(* IEC 61131-3 sources: AXOpen/src/components.ur.robotics/ctrl/src/AxoUrCb3/v_3_x_x, 1 file *)

(* ---- AxoUrCb3.st ---- *)
USING AXOpen.Core;
USING AXOpen.Messaging;
USING AXOpen.Messaging.Static;
USING AXOpen.Components.Robotics;
USING AXOpen.Components.Abstractions.Robotics;
USING Siemens.Simatic.Hardware.Utilities;

NAMESPACE AXOpen.Components.Ur.Robotics.v_3_x_x
    {S7.extern=ReadWrite}
    CLASS AxoUrCb3 EXTENDS AXOpen.Core.AxoComponent IMPLEMENTS AXOpen.Components.Abstractions.Robotics.IAxoRobotics
        VAR PRIVATE
            _infoTimer              :   AXOpen.Timers.OnDelayTimer;
            _errorTimer             :   AXOpen.Timers.OnDelayTimer;
            _context                :   IAxoContext;
            _stopTasksAreActive     :   BOOL;
            _stopType               :   eAxoRoboticsStopType;
            _someTaskIsActive       :   BOOL;

            _initHwCheckDone        :   BOOL;
            _retval                 :   WORD;
            _geoAddr                :   GeoAddr;
            _outHwid                :   UINT;
            _blink                  :   AXOpen.Timers.AxoBlinker;
            _inputsAddress          :   UDINT;
            _inputsCount            :   UINT;
            _outputsAddress         :   UDINT;
            _outputsCount           :   UINT;
        END_VAR

        VAR PUBLIC //HEADER

        END_VAR

        VAR PUBLIC //Tasks
            {#ix-attr:[Container(Layout.Wrap)]}
            {#ix-attr:[ComponentDetails("Tasks")]}
            {#ix-set:AttributeName = "<#Restore#>"}
            RestoreTask : AxoTask;

            {#ix-attr:[ComponentDetails("Tasks")]}
            {#ix-set:AttributeName = "<#Power On Task#>"}
            PowerOnTask : AxoTask;

            {#ix-attr:[Container(Layout.Wrap)]}
            {#ix-attr:[ComponentDetails("Tasks")]}
            {#ix-set:AttributeName = "<#Start at main#>"}
            StartAtMainTask : AxoTask;

            {#ix-attr:[ComponentDetails("Tasks")]}
            {#ix-set:AttributeName = "<#Start motors and program#>"}
            StartMotorsAndProgramTask : AxoTask;

            {#ix-attr:[ComponentDetails("Tasks")]}
            {#ix-set:AttributeName = "<#Stop movements#>"}
            StopMovementsTask : AxoTask;

            {#ix-attr:[ComponentDetails("Tasks")]}
            {#ix-set:AttributeName = "<#Stop movements and program#>"}
            StopMovementsAndProgramTask : AxoTask;

            {#ix-attr:[ComponentDetails("Tasks")]}
            {#ix-set:AttributeName = "<#Start movements with extended parameters#>"}
            StartMovementsTask : AxoTask;

            {#ix-attr:[ComponentDetails("Tasks")]}
            {#ix-set:AttributeName = "<#Start movements with extended parameters#>"}
            MovementParameters : AXOpen.Components.Abstractions.Robotics.AxoRoboticsMovementsParams;
        END_VAR

        VAR PUBLIC //CONFIG
            {#ix-attr:[Container(Layout.Stack)]}
            {#ix-attr:[ComponentDetails("Config")]}
            {#ix-attr:[ReadOnly()]}
            Config  :   AxoUrRobotics_Config;
        END_VAR

        VAR PUBLIC //STATUS
            {#ix-attr:[Container(Layout.Stack)]}
            {#ix-attr:[ComponentDetails("Status")]}
            {#ix-attr:[ReadOnly()]}
            Status         :   AxoUrRobotics_Component_Status;
            {#ix-attr:[ComponentDetails("Status")]}
            {#ix-attr:[ReadOnly()]}
            {#ix-set:AttributeName = "<#Power progress#>"}
            _power_progress  :   INT := 0;
            {#ix-attr:[ComponentDetails("Status")]}
            {#ix-attr:[ReadOnly()]}
            {#ix-set:AttributeName = "<#Movement progress#>"}
            _movement_progress  :   INT := 0;
            Messenger           :   AXOpen.Messaging.Static.AxoMessenger;
            TaskMessenger       :   AXOpen.Messaging.Static.AxoMessenger;
        END_VAR

        VAR PUBLIC //Hardware signals
            {#ix-attr:[ComponentDetails("Hardware signals")]}
            {#ix-attr:[Container(Layout.Wrap)]}
            {#ix-attr:[Group(GroupLayout.GroupBox)]}
            {#ix-set:AttributeName = "<#Inputs#>"}
            {#ix-attr:[ReadOnly()]}
            Inputs              :   AxoUrRobotics_State;
            {#ix-attr:[ComponentDetails("Hardware signals")]}
            {#ix-attr:[Container(Layout.Wrap)]}
            {#ix-attr:[Group(GroupLayout.GroupBox)]}
            {#ix-set:AttributeName = "<#Outputs#>"}
            {#ix-attr:[ReadOnly()]}
            Outputs              :   AxoUrRobotics_Control;
        END_VAR

        VAR PUBLIC //HardwareDiagnostics
            {#ix-attr:[Container(Layout.Stack)]}
            {#ix-attr:[ComponentDetails("Hardware diagnostics")]}
            {#ix-set:AttributeName = "<#Update diagnostics#>"}
            HardwareDiagnosticsTask :   AXOpen.Io.AxoHardwareDiagnostics;
            {#ix-attr:[ComponentDetails("Hardware diagnostics")]}
            {#ix-set:AttributeName = "<#Reboot controller#>"}
            RebootControllerTask : AxoRemoteTask ;
        END_VAR

        ///<summary>
        /// Runs tasks and logic of this component.
        /// >[!IMPORTANT] This method must or one of its overloads be called cyclically.
        ///</summary>
        METHOD PUBLIC Run
            VAR_INPUT
                inParent        :   IAxoObject;
                hwID            :   UINT;
                refPowerOnPulse :   REF_TO BOOL;
            END_VAR
            VAR
                _word : WORD;
                _dword: DWORD;
                _retVal : WORD;
                _data : ARRAY[0..103] OF BYTE;
                _data24 : ARRAY[0..23] OF BYTE;
                _data100 : ARRAY[0..99] OF BYTE;
            END_VAR

            SUPER.Run(inParent);

            Messenger.Serve(THIS);

            IF NOT _initHwCheckDone THEN
                IF inParent = NULL THEN
                    Messenger.Activate(UINT#700, eAxoMessageCategory#ProgrammingError);
                    Status.Error.Id := UINT#700;
                    RETURN;
                END_IF;
                Config.HWIDs.HwId_Device  := hwID;
                IF Config.HWIDs.HwId_Device = UINT#0 THEN
                    Messenger.Activate(UINT#701, eAxoMessageCategory#ProgrammingError);
                    Status.Error.Id := UINT#701;
                    RETURN;
                END_IF;

                _retval := ReadSlotFromHardwareID(hardwareID := Config.HWIDs.HwId_Device, geoAddr :=_geoAddr);
                IF _retval = WORD#8090 THEN
                    Messenger.Activate(UINT#702,eAxoMessageCategory#Error);
                    Status.Error.Id := UINT#702;
                    RETURN;
                END_IF;

                //******************Slot 1*****************//
                _geoAddr.Slot   :=  UINT#1;
                _geoAddr.HardwareType := UINT#4; // (4-Module)
                _retval := ReadHardwareIDFromSlot(geoAddr := _geoAddr, hardwareID => _outHwid);
                IF Config.HWIDs.HwId_AxoUrRobotics_T2O_State = UINT#0 THEN
                    Messenger.Activate(UINT#710,eAxoMessageCategory#Error);
                    Status.Error.Id := UINT#710;
                    RETURN;
                END_IF;
                IF _retval = WORD#8091 THEN
                    Messenger.Activate(UINT#711,eAxoMessageCategory#Error);
                    Status.Error.Id := UINT#711;
                    RETURN;
                END_IF;
                IF _retval = WORD#8094 THEN
                    Messenger.Activate(UINT#712,eAxoMessageCategory#Error);
                    Status.Error.Id := UINT#712;
                    RETURN;
                END_IF;
                IF _retval = WORD#8095 THEN
                    Messenger.Activate(UINT#713,eAxoMessageCategory#Error);
                    Status.Error.Id := UINT#713;
                    RETURN;
                END_IF;
                IF _retval = WORD#8096 THEN
                    Messenger.Activate(UINT#714,eAxoMessageCategory#Error);
                    Status.Error.Id := UINT#714;
                    RETURN;
                END_IF;
                IF _retval = WORD#8097 THEN
                    Messenger.Activate(UINT#715,eAxoMessageCategory#Error);
                    Status.Error.Id := UINT#715;
                    RETURN;
                END_IF;
                ReadHardwareIOAddress(hardwareID := (Config.HWIDs.HwId_AxoUrRobotics_T2O_State) , inputStartAddress => _inputsAddress , inputCount => _inputsCount , outputStartAddress => _outputsAddress , outputCount => _outputsCount);
                IF _inputsCount <> UINT#32 OR _outputsCount <> UINT#0 THEN
                    Messenger.Activate(UINT#716,eAxoMessageCategory#Error);
                    Status.Error.Id := UINT#716;
                    RETURN;
                END_IF;
                //******************Slot 2*****************//
                _geoAddr.Slot   :=  UINT#2;
                _geoAddr.HardwareType := UINT#4; // (4-Module)
                _retval := ReadHardwareIDFromSlot(geoAddr := _geoAddr, hardwareID => _outHwid);
                IF Config.HWIDs.HwId_AxoUrRobotics_T2O_IO = UINT#0 THEN
                    Messenger.Activate(UINT#720,eAxoMessageCategory#Error);
                    Status.Error.Id := UINT#720;
                    RETURN;
                END_IF;
                IF _retval = WORD#8091 THEN
                    Messenger.Activate(UINT#721,eAxoMessageCategory#Error);
                    Status.Error.Id := UINT#721;
                    RETURN;
                END_IF;
                IF _retval = WORD#8094 THEN
                    Messenger.Activate(UINT#722,eAxoMessageCategory#Error);
                    Status.Error.Id := UINT#722;
                    RETURN;
                END_IF;
                IF _retval = WORD#8095 THEN
                    Messenger.Activate(UINT#723,eAxoMessageCategory#Error);
                    Status.Error.Id := UINT#723;
                    RETURN;
                END_IF;
                IF _retval = WORD#8096 THEN
                    Messenger.Activate(UINT#724,eAxoMessageCategory#Error);
                    Status.Error.Id := UINT#724;
                    RETURN;
                END_IF;
                IF _retval = WORD#8097 THEN
                    Messenger.Activate(UINT#725,eAxoMessageCategory#Error);
                    Status.Error.Id := UINT#725;
                    RETURN;
                END_IF;
                ReadHardwareIOAddress(hardwareID := (Config.HWIDs.HwId_AxoUrRobotics_T2O_IO) , inputStartAddress => _inputsAddress , inputCount => _inputsCount , outputStartAddress => _outputsAddress , outputCount => _outputsCount);
                IF _inputsCount <> UINT#68 OR _outputsCount <> UINT#0 THEN
                    Messenger.Activate(UINT#726,eAxoMessageCategory#Error);
                    Status.Error.Id := UINT#726;
                    RETURN;
                END_IF;
                //******************Slot 3*****************//
                _geoAddr.Slot   :=  UINT#3;
                _geoAddr.HardwareType := UINT#4; // (4-Module)
                _retval := ReadHardwareIDFromSlot(geoAddr := _geoAddr, hardwareID => _outHwid);
                IF Config.HWIDs.HwId_AxoUrRobotics_T2O_Joints = UINT#0 THEN
                    Messenger.Activate(UINT#730,eAxoMessageCategory#Error);
                    Status.Error.Id := UINT#730;
                    RETURN;
                END_IF;
                IF _retval = WORD#8091 THEN
                    Messenger.Activate(UINT#731,eAxoMessageCategory#Error);
                    Status.Error.Id := UINT#731;
                    RETURN;
                END_IF;
                IF _retval = WORD#8094 THEN
                    Messenger.Activate(UINT#732,eAxoMessageCategory#Error);
                    Status.Error.Id := UINT#732;
                    RETURN;
                END_IF;
                IF _retval = WORD#8095 THEN
                    Messenger.Activate(UINT#733,eAxoMessageCategory#Error);
                    Status.Error.Id := UINT#733;
                    RETURN;
                END_IF;
                IF _retval = WORD#8096 THEN
                    Messenger.Activate(UINT#734,eAxoMessageCategory#Error);
                    Status.Error.Id := UINT#734;
                    RETURN;
                END_IF;
                IF _retval = WORD#8097 THEN
                    Messenger.Activate(UINT#735,eAxoMessageCategory#Error);
                    Status.Error.Id := UINT#735;
                    RETURN;
                END_IF;
                ReadHardwareIOAddress(hardwareID := (Config.HWIDs.HwId_AxoUrRobotics_T2O_Joints) , inputStartAddress => _inputsAddress , inputCount => _inputsCount , outputStartAddress => _outputsAddress , outputCount => _outputsCount);
                IF _inputsCount <> UINT#104 OR _outputsCount <> UINT#0 THEN
                    Messenger.Activate(UINT#736,eAxoMessageCategory#Error);
                    Status.Error.Id := UINT#736;
                    RETURN;
                END_IF;
                //******************Slot 4*****************//
                _geoAddr.Slot   :=  UINT#4;
                _geoAddr.HardwareType := UINT#4; // (4-Module)
                _retval := ReadHardwareIDFromSlot(geoAddr := _geoAddr, hardwareID => _outHwid);
                IF Config.HWIDs.HwId_AxoUrRobotics_T2O_TCP = UINT#0 THEN
                    Messenger.Activate(UINT#740,eAxoMessageCategory#Error);
                    Status.Error.Id := UINT#740;
                    RETURN;
                END_IF;
                IF _retval = WORD#8091 THEN
                    Messenger.Activate(UINT#741,eAxoMessageCategory#Error);
                    Status.Error.Id := UINT#741;
                    RETURN;
                END_IF;
                IF _retval = WORD#8094 THEN
                    Messenger.Activate(UINT#742,eAxoMessageCategory#Error);
                    Status.Error.Id := UINT#742;
                    RETURN;
                END_IF;
                IF _retval = WORD#8095 THEN
                    Messenger.Activate(UINT#743,eAxoMessageCategory#Error);
                    Status.Error.Id := UINT#743;
                    RETURN;
                END_IF;
                IF _retval = WORD#8096 THEN
                    Messenger.Activate(UINT#744,eAxoMessageCategory#Error);
                    Status.Error.Id := UINT#744;
                    RETURN;
                END_IF;
                IF _retval = WORD#8097 THEN
                    Messenger.Activate(UINT#745,eAxoMessageCategory#Error);
                    Status.Error.Id := UINT#745;
                    RETURN;
                END_IF;
                ReadHardwareIOAddress(hardwareID := (Config.HWIDs.HwId_AxoUrRobotics_T2O_TCP) , inputStartAddress => _inputsAddress , inputCount => _inputsCount , outputStartAddress => _outputsAddress , outputCount => _outputsCount);
                IF _inputsCount <> UINT#76 OR _outputsCount <> UINT#0 THEN
                    Messenger.Activate(UINT#746,eAxoMessageCategory#Error);
                    Status.Error.Id := UINT#746;
                    RETURN;
                END_IF;
                //******************Slot 5*****************//
                _geoAddr.Slot   :=  UINT#5;
                _geoAddr.HardwareType := UINT#4; // (4-Module)
                _retval := ReadHardwareIDFromSlot(geoAddr := _geoAddr, hardwareID => _outHwid);
                IF Config.HWIDs.HwId_AxoUrRobotics_T2O_General_Purpose_Bit_Registers = UINT#0 THEN
                    Messenger.Activate(UINT#750,eAxoMessageCategory#Error);
                    Status.Error.Id := UINT#750;
                    RETURN;
                END_IF;
                IF _retval = WORD#8091 THEN
                    Messenger.Activate(UINT#751,eAxoMessageCategory#Error);
                    Status.Error.Id := UINT#751;
                    RETURN;
                END_IF;
                IF _retval = WORD#8094 THEN
                    Messenger.Activate(UINT#752,eAxoMessageCategory#Error);
                    Status.Error.Id := UINT#752;
                    RETURN;
                END_IF;
                IF _retval = WORD#8095 THEN
                    Messenger.Activate(UINT#753,eAxoMessageCategory#Error);
                    Status.Error.Id := UINT#753;
                    RETURN;
                END_IF;
                IF _retval = WORD#8096 THEN
                    Messenger.Activate(UINT#754,eAxoMessageCategory#Error);
                    Status.Error.Id := UINT#754;
                    RETURN;
                END_IF;
                IF _retval = WORD#8097 THEN
                    Messenger.Activate(UINT#755,eAxoMessageCategory#Error);
                    Status.Error.Id := UINT#755;
                    RETURN;
                END_IF;
                ReadHardwareIOAddress(hardwareID := (Config.HWIDs.HwId_AxoUrRobotics_T2O_General_Purpose_Bit_Registers), inputStartAddress => _inputsAddress , inputCount => _inputsCount , outputStartAddress => _outputsAddress , outputCount => _outputsCount);
                IF _inputsCount <> UINT#8 OR _outputsCount <> UINT#0 THEN
                    Messenger.Activate(UINT#756,eAxoMessageCategory#Error);
                    Status.Error.Id := UINT#756;
                    RETURN;
                END_IF;
                //******************Slot 6*****************//
                _geoAddr.Slot   :=  UINT#6;
                _geoAddr.HardwareType := UINT#4; // (4-Module)
                _retval := ReadHardwareIDFromSlot(geoAddr := _geoAddr, hardwareID => _outHwid);
                IF Config.HWIDs.HwId_AxoUrRobotics_T2O_General_Purpose_Int_Registers = UINT#0 THEN
                    Messenger.Activate(UINT#760,eAxoMessageCategory#Error);
                    Status.Error.Id := UINT#760;
                    RETURN;
                END_IF;
                IF _retval = WORD#8091 THEN
                    Messenger.Activate(UINT#761,eAxoMessageCategory#Error);
                    Status.Error.Id := UINT#761;
                    RETURN;
                END_IF;
                IF _retval = WORD#8094 THEN
                    Messenger.Activate(UINT#762,eAxoMessageCategory#Error);
                    Status.Error.Id := UINT#762;
                    RETURN;
                END_IF;
                IF _retval = WORD#8095 THEN
                    Messenger.Activate(UINT#763,eAxoMessageCategory#Error);
                    Status.Error.Id := UINT#763;
                    RETURN;
                END_IF;
                IF _retval = WORD#8096 THEN
                    Messenger.Activate(UINT#764,eAxoMessageCategory#Error);
                    Status.Error.Id := UINT#764;
                    RETURN;
                END_IF;
                IF _retval = WORD#8097 THEN
                    Messenger.Activate(UINT#765,eAxoMessageCategory#Error);
                    Status.Error.Id := UINT#765;
                    RETURN;
                END_IF;
                ReadHardwareIOAddress(hardwareID := (Config.HWIDs.HwId_AxoUrRobotics_T2O_General_Purpose_Int_Registers), inputStartAddress => _inputsAddress , inputCount => _inputsCount , outputStartAddress => _outputsAddress , outputCount => _outputsCount);
                IF _inputsCount <> UINT#96 OR _outputsCount <> UINT#0 THEN
                    Messenger.Activate(UINT#766,eAxoMessageCategory#Error);
                    Status.Error.Id := UINT#766;
                    RETURN;
                END_IF;
                //******************Slot 7*****************//
                _geoAddr.Slot   :=  UINT#7;
                _geoAddr.HardwareType := UINT#4; // (4-Module)
                _retval := ReadHardwareIDFromSlot(geoAddr := _geoAddr, hardwareID => _outHwid);
                IF Config.HWIDs.HwId_AxoUrRobotics_T2O_General_Purpose_Float_Registers = UINT#0 THEN
                    Messenger.Activate(UINT#770,eAxoMessageCategory#Error);
                    Status.Error.Id := UINT#770;
                    RETURN;
                END_IF;
                IF _retval = WORD#8091 THEN
                    Messenger.Activate(UINT#771,eAxoMessageCategory#Error);
                    Status.Error.Id := UINT#771;
                    RETURN;
                END_IF;
                IF _retval = WORD#8094 THEN
                    Messenger.Activate(UINT#772,eAxoMessageCategory#Error);
                    Status.Error.Id := UINT#772;
                    RETURN;
                END_IF;
                IF _retval = WORD#8095 THEN
                    Messenger.Activate(UINT#773,eAxoMessageCategory#Error);
                    Status.Error.Id := UINT#773;
                    RETURN;
                END_IF;
                IF _retval = WORD#8096 THEN
                    Messenger.Activate(UINT#774,eAxoMessageCategory#Error);
                    Status.Error.Id := UINT#774;
                    RETURN;
                END_IF;
                IF _retval = WORD#8097 THEN
                    Messenger.Activate(UINT#775,eAxoMessageCategory#Error);
                    Status.Error.Id := UINT#775;
                    RETURN;
                END_IF;
                ReadHardwareIOAddress(hardwareID := (Config.HWIDs.HwId_AxoUrRobotics_T2O_General_Purpose_Float_Registers) , inputStartAddress => _inputsAddress , inputCount => _inputsCount , outputStartAddress => _outputsAddress , outputCount => _outputsCount);
                IF _inputsCount <> UINT#132 OR _outputsCount <> UINT#0 THEN
                    Messenger.Activate(UINT#776,eAxoMessageCategory#Error);
                    Status.Error.Id := UINT#776;
                    RETURN;
                END_IF;
                //******************Slot 8*****************//
                _geoAddr.Slot   :=  UINT#8;
                _geoAddr.HardwareType := UINT#4; // (4-Module)
                _retval := ReadHardwareIDFromSlot(geoAddr := _geoAddr, hardwareID => _outHwid);
                IF Config.HWIDs.HwId_AxoUrRobotics_O2T_Robot_IO = UINT#0 THEN
                    Messenger.Activate(UINT#780,eAxoMessageCategory#Error);
                    Status.Error.Id := UINT#780;
                    RETURN;
                END_IF;
                IF _retval = WORD#8091 THEN
                    Messenger.Activate(UINT#781,eAxoMessageCategory#Error);
                    Status.Error.Id := UINT#781;
                    RETURN;
                END_IF;
                IF _retval = WORD#8094 THEN
                    Messenger.Activate(UINT#782,eAxoMessageCategory#Error);
                    Status.Error.Id := UINT#782;
                    RETURN;
                END_IF;
                IF _retval = WORD#8095 THEN
                    Messenger.Activate(UINT#783,eAxoMessageCategory#Error);
                    Status.Error.Id := UINT#783;
                    RETURN;
                END_IF;
                IF _retval = WORD#8096 THEN
                    Messenger.Activate(UINT#784,eAxoMessageCategory#Error);
                    Status.Error.Id := UINT#784;
                    RETURN;
                END_IF;
                IF _retval = WORD#8097 THEN
                    Messenger.Activate(UINT#785,eAxoMessageCategory#Error);
                    Status.Error.Id := UINT#785;
                    RETURN;
                END_IF;
                ReadHardwareIOAddress(hardwareID := (Config.HWIDs.HwId_AxoUrRobotics_O2T_Robot_IO) , inputStartAddress => _inputsAddress , inputCount => _inputsCount , outputStartAddress => _outputsAddress , outputCount => _outputsCount);
                IF _inputsCount <> UINT#0 OR _outputsCount <> UINT#24 THEN
                    Messenger.Activate(UINT#786,eAxoMessageCategory#Error);
                    Status.Error.Id := UINT#786;
                    RETURN;
                END_IF;
                //******************Slot 9*****************//
                _geoAddr.Slot   :=  UINT#9;
                _geoAddr.HardwareType := UINT#4; // (4-Module)
                _retval := ReadHardwareIDFromSlot(geoAddr := _geoAddr, hardwareID => _outHwid);
                IF Config.HWIDs.HwId_AxoUrRobotics_O2T_General_Purpose_Registers_1 = UINT#0 THEN
                    Messenger.Activate(UINT#790,eAxoMessageCategory#Error);
                    Status.Error.Id := UINT#790;
                    RETURN;
                END_IF;
                IF _retval = WORD#8091 THEN
                    Messenger.Activate(UINT#791,eAxoMessageCategory#Error);
                    Status.Error.Id := UINT#791;
                    RETURN;
                END_IF;
                IF _retval = WORD#8094 THEN
                    Messenger.Activate(UINT#792,eAxoMessageCategory#Error);
                    Status.Error.Id := UINT#792;
                    RETURN;
                END_IF;
                IF _retval = WORD#8095 THEN
                    Messenger.Activate(UINT#793,eAxoMessageCategory#Error);
                    Status.Error.Id := UINT#793;
                    RETURN;
                END_IF;
                IF _retval = WORD#8096 THEN
                    Messenger.Activate(UINT#794,eAxoMessageCategory#Error);
                    Status.Error.Id := UINT#794;
                    RETURN;
                END_IF;
                IF _retval = WORD#8097 THEN
                    Messenger.Activate(UINT#795,eAxoMessageCategory#Error);
                    Status.Error.Id := UINT#795;
                    RETURN;
                END_IF;
                ReadHardwareIOAddress(hardwareID := (Config.HWIDs.HwId_AxoUrRobotics_O2T_General_Purpose_Registers_1) , inputStartAddress => _inputsAddress , inputCount => _inputsCount , outputStartAddress => _outputsAddress , outputCount => _outputsCount);
                IF _inputsCount <> UINT#0 OR _outputsCount <> UINT#100 THEN
                    Messenger.Activate(UINT#796,eAxoMessageCategory#Error);
                    Status.Error.Id := UINT#796;
                    RETURN;
                END_IF;
                //******************Slot 10*****************//
                _geoAddr.Slot   :=  UINT#10;
                _geoAddr.HardwareType := UINT#4; // (4-Module)
                _retval := ReadHardwareIDFromSlot(geoAddr := _geoAddr, hardwareID => _outHwid);
                IF Config.HWIDs.HwId_AxoUrRobotics_O2T_General_Purpose_Registers_2 = UINT#0 THEN
                    Messenger.Activate(UINT#800,eAxoMessageCategory#Error);
                    Status.Error.Id := UINT#800;
                    RETURN;
                END_IF;
                IF _retval = WORD#8091 THEN
                    Messenger.Activate(UINT#801,eAxoMessageCategory#Error);
                    Status.Error.Id := UINT#801;
                    RETURN;
                END_IF;
                IF _retval = WORD#8094 THEN
                    Messenger.Activate(UINT#802,eAxoMessageCategory#Error);
                    Status.Error.Id := UINT#802;
                    RETURN;
                END_IF;
                IF _retval = WORD#8095 THEN
                    Messenger.Activate(UINT#803,eAxoMessageCategory#Error);
                    Status.Error.Id := UINT#803;
                    RETURN;
                END_IF;
                IF _retval = WORD#8096 THEN
                    Messenger.Activate(UINT#804,eAxoMessageCategory#Error);
                    Status.Error.Id := UINT#804;
                    RETURN;
                END_IF;
                IF _retval = WORD#8097 THEN
                    Messenger.Activate(UINT#805,eAxoMessageCategory#Error);
                    Status.Error.Id := UINT#805;
                    RETURN;
                END_IF;
                ReadHardwareIOAddress(hardwareID := (Config.HWIDs.HwId_AxoUrRobotics_O2T_General_Purpose_Registers_2) , inputStartAddress => _inputsAddress , inputCount => _inputsCount , outputStartAddress => _outputsAddress , outputCount => _outputsCount);
                IF _inputsCount <> UINT#0 OR _outputsCount <> UINT#100 THEN
                    Messenger.Activate(UINT#806,eAxoMessageCategory#Error);
                    Status.Error.Id := UINT#806;
                    RETURN;
                END_IF;

                IF inParent = NULL THEN
                    Messenger.Activate(UINT#1130,eAxoMessageCategory#Error);
                    Status.Error.Id := UINT#1130;
                    RETURN;
                END_IF;
                IF Config.HWIDs.HwId_Device  = UINT#0 THEN
                    Messenger.Activate(UINT#1131,eAxoMessageCategory#Error);
                    Status.Error.Id := UINT#1131;
                    RETURN;
                END_IF;
                IF Config.HWIDs.HwId_AxoUrRobotics_T2O_State  = UINT#0 THEN
                    Messenger.Activate(UINT#1132,eAxoMessageCategory#Error);
                    Status.Error.Id := UINT#1132;
                    RETURN;
                END_IF;
                IF Config.HWIDs.HwId_AxoUrRobotics_T2O_IO  = UINT#0 THEN
                    Messenger.Activate(UINT#1133,eAxoMessageCategory#Error);
                    Status.Error.Id := UINT#1133;
                    RETURN;
                END_IF;
                IF Config.HWIDs.HwId_AxoUrRobotics_T2O_Joints  = UINT#0 THEN
                    Messenger.Activate(UINT#1134,eAxoMessageCategory#Error);
                    Status.Error.Id := UINT#1134;
                    RETURN;
                END_IF;
                IF Config.HWIDs.HwId_AxoUrRobotics_T2O_TCP  = UINT#0 THEN
                    Messenger.Activate(UINT#1135,eAxoMessageCategory#Error);
                    Status.Error.Id := UINT#1135;
                    RETURN;
                END_IF;
                IF Config.HWIDs.HwId_AxoUrRobotics_T2O_General_Purpose_Bit_Registers  = UINT#0 THEN
                    Messenger.Activate(UINT#1136,eAxoMessageCategory#Error);
                    Status.Error.Id := UINT#1136;
                    RETURN;
                END_IF;
                IF Config.HWIDs.HwId_AxoUrRobotics_T2O_General_Purpose_Int_Registers  = UINT#0 THEN
                    Messenger.Activate(UINT#1137,eAxoMessageCategory#Error);
                    Status.Error.Id := UINT#1137;
                    RETURN;
                END_IF;
                IF Config.HWIDs.HwId_AxoUrRobotics_T2O_General_Purpose_Float_Registers  = UINT#0 THEN
                    Messenger.Activate(UINT#1138,eAxoMessageCategory#Error);
                    Status.Error.Id := UINT#1138;
                    RETURN;
                END_IF;
                IF Config.HWIDs.HwId_AxoUrRobotics_O2T_Robot_IO  = UINT#0 THEN
                    Messenger.Activate(UINT#1139,eAxoMessageCategory#Error);
                    Status.Error.Id := UINT#1139;
                    RETURN;
                END_IF;
                IF Config.HWIDs.HwId_AxoUrRobotics_O2T_General_Purpose_Registers_1  = UINT#0 THEN
                    Messenger.Activate(UINT#1140,eAxoMessageCategory#Error);
                    Status.Error.Id := UINT#1140;
                    RETURN;
                END_IF;
                IF Config.HWIDs.HwId_AxoUrRobotics_O2T_General_Purpose_Registers_2  = UINT#0 THEN
                    Messenger.Activate(UINT#1141,eAxoMessageCategory#Error);
                    Status.Error.Id := UINT#1141;
                    RETURN;
                END_IF;

                _initHwCheckDone    := TRUE;
            END_IF;

            //*******************************************
            _context := THIS.GetContext();

            //*************INITIALIZATION*************
            RestoreTask.Run(THIS);
            PowerOnTask.Run(THIS);
            StopMovementsTask.Run(THIS);
            StopMovementsAndProgramTask.Run(THIS);

            StartAtMainTask.Run(THIS);
            StartMotorsAndProgramTask.Run(THIS);
            StartMovementsTask.Run(THIS);
            HardwareDiagnosticsTask.Run(THIS);
            RebootControllerTask.Run(THIS);

            _stopTasksAreActive := StopMovementsTask.IsBusy() OR StopMovementsAndProgramTask.IsBusy();
            //****************************************
            //********************Diagnostics*********
            HardwareDiagnosticsTask.Run(THIS,Config.HWIDs.HwId_Device);
            RebootControllerTask.Execute(THIS);
            //****************************************
            //*************RESTORE********************
            RestoreTask.SetIsDisabled(FALSE);
            IF RestoreTask.Execute(THIS) THEN
                THIS.Restore();
            END_IF;
            //****************************************

            //***********UPDATE**INPUTS******************
            //Inputs Low level
            //INPUTS T2O STATE ROBOT => st_URO_CB3_T2OInfoData
            _retVal := Siemens.Simatic.DistributedIO.ReadData((Config.HWIDs.HwId_AxoUrRobotics_T2O_State), _data);
            IF _retVal > WORD#0 THEN
                Messenger.Activate(UINT#1201, eAxoMessageCategory#Error);
                Status.Error.Id := UINT#1201;
                RETURN;
            END_IF;
            Inputs.Inputs.Robot.ControllerMajorVersion              := TO_USINT(_data[0]);
            Inputs.Inputs.Robot.ControllerMinorVersion              := TO_USINT(_data[1]);
            Inputs.Inputs.Robot.RobotMode                           := TO_USINT(_data[4]);
            Inputs.Inputs.Robot.RealtimeMachineSeconds              := TO_USINT(_data[5]);
            _word.%B1                                               := _data[6];
            _word.%B0                                               := _data[7];
            Inputs.Inputs.Robot.RealtimeMachineMilliseconds         := TO_UINT(_word);
            Inputs.Inputs.Robot.RealtimeMachineMinutes              := TO_USINT(_data[8]);
            Inputs.Inputs.Robot.RealtimeMachineHours                := TO_USINT(_data[9]);
            _word.%B1                                               := _data[10];
            _word.%B0                                               := _data[11];
            Inputs.Inputs.Robot.RealtimeMachineDays                 := TO_UINT(_word);
            _dword.%B3                                              := _data[12];
            _dword.%B2                                              := _data[13];
            _dword.%B1                                              := _data[14];
            _dword.%B0                                              := _data[15];
            Inputs.Inputs.Robot.RobotCurrent                        := TO_REAL(_dword);
            //INPUTS T2O STATE ROBOT => st_URO_CB3_T2OStateData
            Inputs.Inputs.Robot.PW_IsPowerOn                        := _data[16].%X0;
            Inputs.Inputs.Robot.PR_IsProgramRunning                 := _data[16].%X1;
            Inputs.Inputs.Robot.TB_IsTeachButtonPressed             := _data[16].%X2;
            Inputs.Inputs.Robot.PB_IsPowerButtonPressed             := _data[16].%X3;
            _dword.%B3                                              := _data[20];
            _dword.%B2                                              := _data[21];
            _dword.%B1                                              := _data[22];
            _dword.%B0                                              := _data[23];
            Inputs.Inputs.Robot.SpeedSliderFraction                 := REAL#100.0 * TO_REAL(_dword);
            Inputs.Inputs.Safety.SafetyMode                         := TO_USINT(_data[24]);
            Inputs.Inputs.Safety.NO_IsNormalMode                    := _data[28].%X0;
            Inputs.Inputs.Safety.RD_IsReducedMode                   := _data[28].%X1;
            Inputs.Inputs.Safety.PS_IsProtectiveStopped             := _data[28].%X2;
            Inputs.Inputs.Safety.RC_IsRecoveryMode                  := _data[28].%X3;
            Inputs.Inputs.Safety.SS_IsSafeguardStopped              := _data[28].%X4;
            Inputs.Inputs.Safety.SES_IsSystemEmergencyStopped       := _data[28].%X5;
            Inputs.Inputs.Safety.RES_IsRobotEmergencyStopped        := _data[28].%X6;
            Inputs.Inputs.Safety.ES_IsEmergencyStopped              := _data[28].%X7;
            Inputs.Inputs.Safety.VL_IsViolation                     := _data[29].%X0;
            Inputs.Inputs.Safety.FT_IsFault                         := _data[29].%X1;
            Inputs.Inputs.Safety.ST_IsStoppedDueSafety              := _data[29].%X2;

            //INPUTS T20 IO => st_URO_CB3_T2OIoStateData
            _retVal := Siemens.Simatic.DistributedIO.ReadData((Config.HWIDs.HwId_AxoUrRobotics_T2O_IO), _data);
            IF _retVal > WORD#0 THEN
                Messenger.Activate(UINT#1202, eAxoMessageCategory#Error);
                Status.Error.Id := UINT#1202;
                RETURN;
            END_IF;
            Inputs.Inputs.IO.StandardDigitalInputs                  := TO_USINT(_data[0]);
            Inputs.Inputs.IO.ConfigurableDigitalInputs              := TO_USINT(_data[1]);
            Inputs.Inputs.IO.StandardDigitalOutputs                 := TO_USINT(_data[2]);
            Inputs.Inputs.IO.ConfigurableDigitalOutputs             := TO_USINT(_data[3]);
            Inputs.Inputs.IO.AnalogIoTypes                          := TO_USINT(_data[4]);
            _dword.%B3                                              := _data[8];
            _dword.%B2                                              := _data[9];
            _dword.%B1                                              := _data[10];
            _dword.%B0                                              := _data[11];
            Inputs.Inputs.IO.StandardAnalogInput_0                  := TO_REAL(_dword);
            _dword.%B3                                              := _data[12];
            _dword.%B2                                              := _data[13];
            _dword.%B1                                              := _data[14];
            _dword.%B0                                              := _data[15];
            Inputs.Inputs.IO.StandardAnalogInput_1                  := TO_REAL(_dword);
            _dword.%B3                                              := _data[16];
            _dword.%B2                                              := _data[17];
            _dword.%B1                                              := _data[18];
            _dword.%B0                                              := _data[19];
            Inputs.Inputs.IO.StandardAnalogOutput_0                 := TO_REAL(_dword);
            _dword.%B3                                              := _data[20];
            _dword.%B2                                              := _data[21];
            _dword.%B1                                              := _data[22];
            _dword.%B0                                              := _data[23];
            Inputs.Inputs.IO.StandardAnalogOutput_1                 := TO_REAL(_dword);
            _dword.%B3                                              := _data[24];
            _dword.%B2                                              := _data[25];
            _dword.%B1                                              := _data[26];
            _dword.%B0                                              := _data[27];
            Inputs.Inputs.IO.Current                                := TO_REAL(_dword);

            Inputs.Inputs.IO.Euromap67InputBit_0                    := _data[28].%X0;
            Inputs.Inputs.IO.Euromap67InputBit_1                    := _data[28].%X1;
            Inputs.Inputs.IO.Euromap67InputBit_2                    := _data[28].%X2;
            Inputs.Inputs.IO.Euromap67InputBit_3                    := _data[28].%X3;
            Inputs.Inputs.IO.Euromap67InputBit_4                    := _data[28].%X4;
            Inputs.Inputs.IO.Euromap67InputBit_5                    := _data[28].%X5;
            Inputs.Inputs.IO.Euromap67InputBit_6                    := _data[28].%X6;
            Inputs.Inputs.IO.Euromap67InputBit_7                    := _data[28].%X7;
            Inputs.Inputs.IO.Euromap67InputBit_8                    := _data[29].%X0;
            Inputs.Inputs.IO.Euromap67InputBit_9                    := _data[29].%X1;
            Inputs.Inputs.IO.Euromap67InputBit_10                   := _data[29].%X2;
            Inputs.Inputs.IO.Euromap67InputBit_11                   := _data[29].%X3;
            Inputs.Inputs.IO.Euromap67InputBit_12                   := _data[29].%X4;
            Inputs.Inputs.IO.Euromap67InputBit_13                   := _data[29].%X5;
            Inputs.Inputs.IO.Euromap67InputBit_14                   := _data[29].%X6;
            Inputs.Inputs.IO.Euromap67InputBit_15                   := _data[29].%X7;
            Inputs.Inputs.IO.Euromap67InputBit_16                   := _data[30].%X0;
            Inputs.Inputs.IO.Euromap67InputBit_17                   := _data[30].%X1;
            Inputs.Inputs.IO.Euromap67InputBit_18                   := _data[30].%X2;
            Inputs.Inputs.IO.Euromap67InputBit_19                   := _data[30].%X3;
            Inputs.Inputs.IO.Euromap67InputBit_20                   := _data[30].%X4;
            Inputs.Inputs.IO.Euromap67InputBit_21                   := _data[30].%X5;
            Inputs.Inputs.IO.Euromap67InputBit_22                   := _data[30].%X6;
            Inputs.Inputs.IO.Euromap67InputBit_23                   := _data[30].%X7;
            Inputs.Inputs.IO.Euromap67InputBit_24                   := _data[31].%X0;
            Inputs.Inputs.IO.Euromap67InputBit_25                   := _data[31].%X1;
            Inputs.Inputs.IO.Euromap67InputBit_26                   := _data[31].%X2;
            Inputs.Inputs.IO.Euromap67InputBit_27                   := _data[31].%X3;
            Inputs.Inputs.IO.Euromap67InputBit_28                   := _data[31].%X4;
            Inputs.Inputs.IO.Euromap67InputBit_29                   := _data[31].%X5;
            Inputs.Inputs.IO.Euromap67InputBit_30                   := _data[31].%X6;
            Inputs.Inputs.IO.Euromap67InputBit_31                   := _data[31].%X7;

            Inputs.Inputs.IO.Euromap67OutputBit_0                   := _data[32].%X0;
            Inputs.Inputs.IO.Euromap67OutputBit_1                   := _data[32].%X1;
            Inputs.Inputs.IO.Euromap67OutputBit_2                   := _data[32].%X2;
            Inputs.Inputs.IO.Euromap67OutputBit_3                   := _data[32].%X3;
            Inputs.Inputs.IO.Euromap67OutputBit_4                   := _data[32].%X4;
            Inputs.Inputs.IO.Euromap67OutputBit_5                   := _data[32].%X5;
            Inputs.Inputs.IO.Euromap67OutputBit_6                   := _data[32].%X6;
            Inputs.Inputs.IO.Euromap67OutputBit_7                   := _data[32].%X7;
            Inputs.Inputs.IO.Euromap67OutputBit_8                   := _data[33].%X0;
            Inputs.Inputs.IO.Euromap67OutputBit_9                   := _data[33].%X1;
            Inputs.Inputs.IO.Euromap67OutputBit_10                  := _data[33].%X2;
            Inputs.Inputs.IO.Euromap67OutputBit_11                  := _data[33].%X3;
            Inputs.Inputs.IO.Euromap67OutputBit_12                  := _data[33].%X4;
            Inputs.Inputs.IO.Euromap67OutputBit_13                  := _data[33].%X5;
            Inputs.Inputs.IO.Euromap67OutputBit_14                  := _data[33].%X6;
            Inputs.Inputs.IO.Euromap67OutputBit_15                  := _data[33].%X7;
            Inputs.Inputs.IO.Euromap67OutputBit_16                  := _data[34].%X0;
            Inputs.Inputs.IO.Euromap67OutputBit_17                  := _data[34].%X1;
            Inputs.Inputs.IO.Euromap67OutputBit_18                  := _data[34].%X2;
            Inputs.Inputs.IO.Euromap67OutputBit_19                  := _data[34].%X3;
            Inputs.Inputs.IO.Euromap67OutputBit_20                  := _data[34].%X4;
            Inputs.Inputs.IO.Euromap67OutputBit_21                  := _data[34].%X5;
            Inputs.Inputs.IO.Euromap67OutputBit_22                  := _data[34].%X6;
            Inputs.Inputs.IO.Euromap67OutputBit_23                  := _data[34].%X7;
            Inputs.Inputs.IO.Euromap67OutputBit_24                  := _data[35].%X0;
            Inputs.Inputs.IO.Euromap67OutputBit_25                  := _data[35].%X1;
            Inputs.Inputs.IO.Euromap67OutputBit_26                  := _data[35].%X2;
            Inputs.Inputs.IO.Euromap67OutputBit_27                  := _data[35].%X3;
            Inputs.Inputs.IO.Euromap67OutputBit_28                  := _data[35].%X4;
            Inputs.Inputs.IO.Euromap67OutputBit_29                  := _data[35].%X5;
            Inputs.Inputs.IO.Euromap67OutputBit_30                  := _data[35].%X6;
            Inputs.Inputs.IO.Euromap67OutputBit_31                  := _data[35].%X7;

            _dword.%B3                                              := _data[36];
            _dword.%B2                                              := _data[37];
            _dword.%B1                                              := _data[38];
            _dword.%B0                                              := _data[39];
            Inputs.Inputs.IO.Euromap6724Voltage                     := TO_REAL(_dword);

            _dword.%B3                                              := _data[40];
            _dword.%B2                                              := _data[41];
            _dword.%B1                                              := _data[42];
            _dword.%B0                                              := _data[43];
            Inputs.Inputs.IO.Euromap6724VCurrent                    := TO_REAL(_dword);

            //INPUTS T20 IO => st_URO_CB3_T2OToolStateData
            Inputs.Inputs.Tool.ToolMode                             := TO_USINT(_data[44]);
            Inputs.Inputs.Tool.TDI_ToolDigitalInputs                := TO_USINT(_data[45]);
            Inputs.Inputs.Tool.TDO_ToolDigitalOutputs               := TO_USINT(_data[46]);
            Inputs.Inputs.Tool.TAIT_ToolAnalogInputTypes            := TO_USINT(_data[47]);

            _dword.%B3                                              := _data[48];
            _dword.%B2                                              := _data[49];
            _dword.%B1                                              := _data[50];
            _dword.%B0                                              := _data[51];
            Inputs.Inputs.Tool.ToolAnalogInput_0                    := TO_REAL(_dword);

            _dword.%B3                                              := _data[52];
            _dword.%B2                                              := _data[53];
            _dword.%B1                                              := _data[54];
            _dword.%B0                                              := _data[55];
            Inputs.Inputs.Tool.ToolAnalogInput_1                    := TO_REAL(_dword);

            _dword.%B3                                              := _data[56];
            _dword.%B2                                              := _data[57];
            _dword.%B1                                              := _data[58];
            _dword.%B0                                              := _data[59];
            Inputs.Inputs.Tool.ToolOutputVoltage                    := TO_REAL(_dword);

            _dword.%B3                                              := _data[60];
            _dword.%B2                                              := _data[61];
            _dword.%B1                                              := _data[62];
            _dword.%B0                                              := _data[63];
            Inputs.Inputs.Tool.ToolCurrent                          := TO_REAL(_dword);

            // //INPUTS T20 JOINT => st_URO_CB3_T2OJointsData
            _retVal := Siemens.Simatic.DistributedIO.ReadData((Config.HWIDs.HwId_AxoUrRobotics_T2O_Joints), _data);
            IF _retVal > WORD#0 THEN
                Messenger.Activate(UINT#1203, eAxoMessageCategory#Error);
                Status.Error.Id := UINT#1203;
                RETURN;
            END_IF;
            _dword.%B3                                              := _data[0];
            _dword.%B2                                              := _data[1];
            _dword.%B1                                              := _data[2];
            _dword.%B0                                              := _data[3];
            Inputs.Inputs.Joints.JointPosition_0                    := REAL#57.2957795 * TO_REAL(_dword);

            _dword.%B3                                              := _data[4];
            _dword.%B2                                              := _data[5];
            _dword.%B1                                              := _data[6];
            _dword.%B0                                              := _data[7];
            Inputs.Inputs.Joints.JointPosition_1                    := REAL#57.2957795 * TO_REAL(_dword);

            _dword.%B3                                              := _data[8];
            _dword.%B2                                              := _data[9];
            _dword.%B1                                              := _data[10];
            _dword.%B0                                              := _data[11];
            Inputs.Inputs.Joints.JointPosition_2                    := REAL#57.2957795 * TO_REAL(_dword);

            _dword.%B3                                              := _data[12];
            _dword.%B2                                              := _data[13];
            _dword.%B1                                              := _data[14];
            _dword.%B0                                              := _data[15];
            Inputs.Inputs.Joints.JointPosition_3                    := REAL#57.2957795 * TO_REAL(_dword);

            _dword.%B3                                              := _data[16];
            _dword.%B2                                              := _data[17];
            _dword.%B1                                              := _data[18];
            _dword.%B0                                              := _data[19];
            Inputs.Inputs.Joints.JointPosition_4                    := REAL#57.2957795 * TO_REAL(_dword);

            _dword.%B3                                              := _data[20];
            _dword.%B2                                              := _data[21];
            _dword.%B1                                              := _data[22];
            _dword.%B0                                              := _data[23];
            Inputs.Inputs.Joints.JointPosition_5                    := REAL#57.2957795 * TO_REAL(_dword);

            _dword.%B3                                              := _data[24];
            _dword.%B2                                              := _data[25];
            _dword.%B1                                              := _data[26];
            _dword.%B0                                              := _data[27];
            Inputs.Inputs.Joints.JointVelocity_0                    :=  TO_REAL(_dword);

            _dword.%B3                                              := _data[28];
            _dword.%B2                                              := _data[29];
            _dword.%B1                                              := _data[30];
            _dword.%B0                                              := _data[31];
            Inputs.Inputs.Joints.JointVelocity_1                    :=  TO_REAL(_dword);

            _dword.%B3                                              := _data[32];
            _dword.%B2                                              := _data[33];
            _dword.%B1                                              := _data[34];
            _dword.%B0                                              := _data[35];
            Inputs.Inputs.Joints.JointVelocity_2                    :=  TO_REAL(_dword);

            _dword.%B3                                              := _data[36];
            _dword.%B2                                              := _data[37];
            _dword.%B1                                              := _data[38];
            _dword.%B0                                              := _data[39];
            Inputs.Inputs.Joints.JointVelocity_3                    :=  TO_REAL(_dword);

            _dword.%B3                                              := _data[40];
            _dword.%B2                                              := _data[41];
            _dword.%B1                                              := _data[42];
            _dword.%B0                                              := _data[43];
            Inputs.Inputs.Joints.JointVelocity_4                    :=  TO_REAL(_dword);

            _dword.%B3                                              := _data[44];
            _dword.%B2                                              := _data[45];
            _dword.%B1                                              := _data[46];
            _dword.%B0                                              := _data[47];
            Inputs.Inputs.Joints.JointVelocity_5                    :=  TO_REAL(_dword);

            _dword.%B3                                              := _data[48];
            _dword.%B2                                              := _data[49];
            _dword.%B1                                              := _data[50];
            _dword.%B0                                              := _data[51];
            Inputs.Inputs.Joints.JointCurrent_0                     :=  TO_REAL(_dword);

            _dword.%B3                                              := _data[52];
            _dword.%B2                                              := _data[53];
            _dword.%B1                                              := _data[54];
            _dword.%B0                                              := _data[55];
            Inputs.Inputs.Joints.JointCurrent_1                     :=  TO_REAL(_dword);

            _dword.%B3                                              := _data[56];
            _dword.%B2                                              := _data[57];
            _dword.%B1                                              := _data[58];
            _dword.%B0                                              := _data[59];
            Inputs.Inputs.Joints.JointCurrent_2                     :=  TO_REAL(_dword);

            _dword.%B3                                              := _data[60];
            _dword.%B2                                              := _data[61];
            _dword.%B1                                              := _data[62];
            _dword.%B0                                              := _data[63];
            Inputs.Inputs.Joints.JointCurrent_3                     :=  TO_REAL(_dword);

            _dword.%B3                                              := _data[64];
            _dword.%B2                                              := _data[65];
            _dword.%B1                                              := _data[66];
            _dword.%B0                                              := _data[67];
            Inputs.Inputs.Joints.JointCurrent_4                     :=  TO_REAL(_dword);

            _dword.%B3                                              := _data[68];
            _dword.%B2                                              := _data[69];
            _dword.%B1                                              := _data[70];
            _dword.%B0                                              := _data[71];
            Inputs.Inputs.Joints.JointCurrent_5                     :=  TO_REAL(_dword);

            _dword.%B3                                              := _data[72];
            _dword.%B2                                              := _data[73];
            _dword.%B1                                              := _data[74];
            _dword.%B0                                              := _data[75];
            Inputs.Inputs.Joints.JointTemperature_0                 :=  TO_REAL(_dword);

            _dword.%B3                                              := _data[76];
            _dword.%B2                                              := _data[77];
            _dword.%B1                                              := _data[78];
            _dword.%B0                                              := _data[79];
            Inputs.Inputs.Joints.JointTemperature_1                 :=  TO_REAL(_dword);

            _dword.%B3                                              := _data[80];
            _dword.%B2                                              := _data[81];
            _dword.%B1                                              := _data[82];
            _dword.%B0                                              := _data[83];
            Inputs.Inputs.Joints.JointTemperature_2                 :=  TO_REAL(_dword);

            _dword.%B3                                              := _data[84];
            _dword.%B2                                              := _data[85];
            _dword.%B1                                              := _data[86];
            _dword.%B0                                              := _data[87];
            Inputs.Inputs.Joints.JointTemperature_3                 :=  TO_REAL(_dword);

            _dword.%B3                                              := _data[88];
            _dword.%B2                                              := _data[89];
            _dword.%B1                                              := _data[90];
            _dword.%B0                                              := _data[91];
            Inputs.Inputs.Joints.JointTemperature_4                 :=  TO_REAL(_dword);

            _dword.%B3                                              := _data[92];
            _dword.%B2                                              := _data[93];
            _dword.%B1                                              := _data[94];
            _dword.%B0                                              := _data[95];
            Inputs.Inputs.Joints.JointTemperature_5                 :=  TO_REAL(_dword);

            Inputs.Inputs.Joints.JointMode_0                        := TO_USINT(_data[96]);
            Inputs.Inputs.Joints.JointMode_1                        := TO_USINT(_data[97]);
            Inputs.Inputs.Joints.JointMode_2                        := TO_USINT(_data[98]);
            Inputs.Inputs.Joints.JointMode_3                        := TO_USINT(_data[99]);
            Inputs.Inputs.Joints.JointMode_4                        := TO_USINT(_data[100]);
            Inputs.Inputs.Joints.JointMode_5                        := TO_USINT(_data[101]);

            //INPUTS T20 TCP => st_URO_CB3_T2OTcpData
            _retVal := Siemens.Simatic.DistributedIO.ReadData((Config.HWIDs.HwId_AxoUrRobotics_T2O_TCP), _data);
            IF _retVal > WORD#0 THEN
                Messenger.Activate(UINT#1204, eAxoMessageCategory#Error);
                Status.Error.Id := UINT#1204;
                RETURN;
            END_IF;
            _dword.%B3                                              := _data[0];
            _dword.%B2                                              := _data[1];
            _dword.%B1                                              := _data[2];
            _dword.%B0                                              := _data[3];
            Inputs.Inputs.TCP.Postition.X                           := REAL#1000.0 * TO_REAL(_dword);

            _dword.%B3                                              := _data[4];
            _dword.%B2                                              := _data[5];
            _dword.%B1                                              := _data[6];
            _dword.%B0                                              := _data[7];
            Inputs.Inputs.TCP.Postition.Y                           := REAL#1000.0 * TO_REAL(_dword);

            _dword.%B3                                              := _data[8];
            _dword.%B2                                              := _data[9];
            _dword.%B1                                              := _data[10];
            _dword.%B0                                              := _data[11];
            Inputs.Inputs.TCP.Postition.Z                           := REAL#1000.0 * TO_REAL(_dword);

            _dword.%B3                                              := _data[12];
            _dword.%B2                                              := _data[13];
            _dword.%B1                                              := _data[14];
            _dword.%B0                                              := _data[15];
            Inputs.Inputs.TCP.Postition.Rx                          := TO_REAL(_dword);

            _dword.%B3                                              := _data[16];
            _dword.%B2                                              := _data[17];
            _dword.%B1                                              := _data[18];
            _dword.%B0                                              := _data[19];
            Inputs.Inputs.TCP.Postition.Ry                          := TO_REAL(_dword);

            _dword.%B3                                              := _data[20];
            _dword.%B2                                              := _data[21];
            _dword.%B1                                              := _data[22];
            _dword.%B0                                              := _data[23];
            Inputs.Inputs.TCP.Postition.Rz                          := TO_REAL(_dword);

            _dword.%B3                                              := _data[24];
            _dword.%B2                                              := _data[25];
            _dword.%B1                                              := _data[26];
            _dword.%B0                                              := _data[27];
            Inputs.Inputs.TCP.Velocity.X                            := REAL#1000.0 * TO_REAL(_dword);

            _dword.%B3                                              := _data[28];
            _dword.%B2                                              := _data[29];
            _dword.%B1                                              := _data[30];
            _dword.%B0                                              := _data[31];
            Inputs.Inputs.TCP.Velocity.Y                            := REAL#1000.0 * TO_REAL(_dword);

            _dword.%B3                                              := _data[32];
            _dword.%B2                                              := _data[33];
            _dword.%B1                                              := _data[34];
            _dword.%B0                                              := _data[35];
            Inputs.Inputs.TCP.Velocity.Z                            := REAL#1000.0 * TO_REAL(_dword);

            _dword.%B3                                              := _data[36];
            _dword.%B2                                              := _data[37];
            _dword.%B1                                              := _data[38];
            _dword.%B0                                              := _data[39];
            Inputs.Inputs.TCP.Velocity.Rx                           := TO_REAL(_dword);

            _dword.%B3                                              := _data[40];
            _dword.%B2                                              := _data[41];
            _dword.%B1                                              := _data[42];
            _dword.%B0                                              := _data[43];
            Inputs.Inputs.TCP.Velocity.Ry                           := TO_REAL(_dword);

            _dword.%B3                                              := _data[44];
            _dword.%B2                                              := _data[45];
            _dword.%B1                                              := _data[46];
            _dword.%B0                                              := _data[47];
            Inputs.Inputs.TCP.Velocity.Rz                           := TO_REAL(_dword);

            _dword.%B3                                              := _data[48];
            _dword.%B2                                              := _data[49];
            _dword.%B1                                              := _data[50];
            _dword.%B0                                              := _data[51];
            Inputs.Inputs.TCP.Force.X                               := TO_REAL(_dword);

            _dword.%B3                                              := _data[52];
            _dword.%B2                                              := _data[53];
            _dword.%B1                                              := _data[54];
            _dword.%B0                                              := _data[55];
            Inputs.Inputs.TCP.Force.Y                               := TO_REAL(_dword);

            _dword.%B3                                              := _data[56];
            _dword.%B2                                              := _data[57];
            _dword.%B1                                              := _data[58];
            _dword.%B0                                              := _data[59];
            Inputs.Inputs.TCP.Force.Z                               := TO_REAL(_dword);

            _dword.%B3                                              := _data[60];
            _dword.%B2                                              := _data[61];
            _dword.%B1                                              := _data[62];
            _dword.%B0                                              := _data[63];
            Inputs.Inputs.TCP.Torque.X                              := TO_REAL(_dword);

            _dword.%B3                                              := _data[64];
            _dword.%B2                                              := _data[65];
            _dword.%B1                                              := _data[66];
            _dword.%B0                                              := _data[67];
            Inputs.Inputs.TCP.Torque.Y                              := TO_REAL(_dword);

            _dword.%B3                                              := _data[68];
            _dword.%B2                                              := _data[69];
            _dword.%B1                                              := _data[70];
            _dword.%B0                                              := _data[71];
            Inputs.Inputs.TCP.Torque.Z                              := TO_REAL(_dword);

            _dword.%B3                                              := _data[72];
            _dword.%B2                                              := _data[73];
            _dword.%B1                                              := _data[74];
            _dword.%B0                                              := _data[75];
            Inputs.Inputs.TCP.TCP_ForceScalar                       := TO_REAL(_dword);

            //INPUTS T20 BITS => st_URO_CB3_T2OBitRegsData
            _retVal := Siemens.Simatic.DistributedIO.ReadData((Config.HWIDs.HwId_AxoUrRobotics_T2O_General_Purpose_Bit_Registers), _data);
            IF _retVal > WORD#0 THEN
                Messenger.Activate(UINT#1205, eAxoMessageCategory#Error);
                Status.Error.Id := UINT#1205;
                RETURN;
            END_IF;
            Inputs.Inputs.Bits.Register_0                           := _data[0].%X0;
            Inputs.Inputs.Bits.Register_1                           := _data[0].%X1;
            Inputs.Inputs.Bits.Register_2                           := _data[0].%X2;
            Inputs.Inputs.Bits.Register_3                           := _data[0].%X3;
            Inputs.Inputs.Bits.Register_4                           := _data[0].%X4;
            Inputs.Inputs.Bits.Register_5                           := _data[0].%X5;
            Inputs.Inputs.Bits.Register_6                           := _data[0].%X6;
            Inputs.Inputs.Bits.Register_7                           := _data[0].%X7;

            Inputs.Inputs.Bits.Register_8                           := _data[1].%X0;
            Inputs.Inputs.Bits.Register_9                           := _data[1].%X1;
            Inputs.Inputs.Bits.Register_10                          := _data[1].%X2;
            Inputs.Inputs.Bits.Register_11                          := _data[1].%X3;
            Inputs.Inputs.Bits.Register_12                          := _data[1].%X4;
            Inputs.Inputs.Bits.Register_13                          := _data[1].%X5;
            Inputs.Inputs.Bits.Register_14                          := _data[1].%X6;
            Inputs.Inputs.Bits.Register_15                          := _data[1].%X7;

            Inputs.Inputs.Bits.Register_16                          := _data[2].%X0;
            Inputs.Inputs.Bits.Register_17                          := _data[2].%X1;
            Inputs.Inputs.Bits.Register_18                          := _data[2].%X2;
            Inputs.Inputs.Bits.Register_19                          := _data[2].%X3;
            Inputs.Inputs.Bits.Register_20                          := _data[2].%X4;
            Inputs.Inputs.Bits.Register_21                          := _data[2].%X5;
            Inputs.Inputs.Bits.Register_22                          := _data[2].%X6;
            Inputs.Inputs.Bits.Register_23                          := _data[2].%X7;

            Inputs.Inputs.Bits.Register_24                          := _data[3].%X0;
            Inputs.Inputs.Bits.Register_25                          := _data[3].%X1;
            Inputs.Inputs.Bits.Register_26                          := _data[3].%X2;
            Inputs.Inputs.Bits.Register_27                          := _data[3].%X3;
            Inputs.Inputs.Bits.Register_28                          := _data[3].%X4;
            Inputs.Inputs.Bits.Register_29                          := _data[3].%X5;
            Inputs.Inputs.Bits.Register_30                          := _data[3].%X6;
            Inputs.Inputs.Bits.Register_31                          := _data[3].%X7;

            Inputs.Inputs.Bits.Register_32                          := _data[4].%X0;
            Inputs.Inputs.Bits.Register_33                          := _data[4].%X1;
            Inputs.Inputs.Bits.Register_34                          := _data[4].%X2;
            Inputs.Inputs.Bits.Register_35                          := _data[4].%X3;
            Inputs.Inputs.Bits.Register_36                          := _data[4].%X4;
            Inputs.Inputs.Bits.Register_37                          := _data[4].%X5;
            Inputs.Inputs.Bits.Register_38                          := _data[4].%X6;
            Inputs.Inputs.Bits.Register_39                          := _data[4].%X7;

            Inputs.Inputs.Bits.Register_40                          := _data[5].%X0;
            Inputs.Inputs.Bits.Register_41                          := _data[5].%X1;
            Inputs.Inputs.Bits.Register_42                          := _data[5].%X2;
            Inputs.Inputs.Bits.Register_43                          := _data[5].%X3;
            Inputs.Inputs.Bits.Register_44                          := _data[5].%X4;
            Inputs.Inputs.Bits.Register_45                          := _data[5].%X5;
            Inputs.Inputs.Bits.Register_46                          := _data[5].%X6;
            Inputs.Inputs.Bits.Register_47                          := _data[5].%X7;

            Inputs.Inputs.Bits.Register_48                          := _data[6].%X0;
            Inputs.Inputs.Bits.Register_49                          := _data[6].%X1;
            Inputs.Inputs.Bits.Register_50                          := _data[6].%X2;
            Inputs.Inputs.Bits.Register_51                          := _data[6].%X3;
            Inputs.Inputs.Bits.Register_52                          := _data[6].%X4;
            Inputs.Inputs.Bits.Register_53                          := _data[6].%X5;
            Inputs.Inputs.Bits.Register_54                          := _data[6].%X6;
            Inputs.Inputs.Bits.Register_55                          := _data[6].%X7;

            Inputs.Inputs.Bits.Register_56                          := _data[7].%X0;
            Inputs.Inputs.Bits.Register_57                          := _data[7].%X1;
            Inputs.Inputs.Bits.Register_58                          := _data[7].%X2;
            Inputs.Inputs.Bits.Register_59                          := _data[7].%X3;
            Inputs.Inputs.Bits.Register_60                          := _data[7].%X4;
            Inputs.Inputs.Bits.Register_61                          := _data[7].%X5;
            Inputs.Inputs.Bits.Register_62                          := _data[7].%X6;
            Inputs.Inputs.Bits.Register_63                          := _data[7].%X7;

            //INPUTS T20 BITS => st_URO_CB3_T2OIntRegsData
            _retVal := Siemens.Simatic.DistributedIO.ReadData((Config.HWIDs.HwId_AxoUrRobotics_T2O_General_Purpose_Int_Registers), _data);
            IF _retVal > WORD#0 THEN
                Messenger.Activate(UINT#1206, eAxoMessageCategory#Error);
                Status.Error.Id := UINT#1206;
                RETURN;
            END_IF;
            _dword.%B3                                              := _data[0];
            _dword.%B2                                              := _data[1];
            _dword.%B1                                              := _data[2];
            _dword.%B0                                              := _data[3];
            Inputs.Inputs.Ints.Register_0                           := TO_DINT(_dword);

            _dword.%B3                                              := _data[4];
            _dword.%B2                                              := _data[5];
            _dword.%B1                                              := _data[6];
            _dword.%B0                                              := _data[7];
            Inputs.Inputs.Ints.Register_1                           := TO_DINT(_dword);

            _dword.%B3                                              := _data[8];
            _dword.%B2                                              := _data[9];
            _dword.%B1                                              := _data[10];
            _dword.%B0                                              := _data[11];
            Inputs.Inputs.Ints.Register_2                           := TO_DINT(_dword);

            _dword.%B3                                              := _data[12];
            _dword.%B2                                              := _data[13];
            _dword.%B1                                              := _data[14];
            _dword.%B0                                              := _data[15];
            Inputs.Inputs.Ints.Register_3                           := TO_DINT(_dword);

            _dword.%B3                                              := _data[16];
            _dword.%B2                                              := _data[17];
            _dword.%B1                                              := _data[18];
            _dword.%B0                                              := _data[19];
            Inputs.Inputs.Ints.Register_4                           := TO_DINT(_dword);

            _dword.%B3                                              := _data[20];
            _dword.%B2                                              := _data[21];
            _dword.%B1                                              := _data[22];
            _dword.%B0                                              := _data[23];
            Inputs.Inputs.Ints.Register_5                           := TO_DINT(_dword);

            _dword.%B3                                              := _data[24];
            _dword.%B2                                              := _data[25];
            _dword.%B1                                              := _data[26];
            _dword.%B0                                              := _data[27];
            Inputs.Inputs.Ints.Register_6                           := TO_DINT(_dword);

            _dword.%B3                                              := _data[28];
            _dword.%B2                                              := _data[29];
            _dword.%B1                                              := _data[30];
            _dword.%B0                                              := _data[31];
            Inputs.Inputs.Ints.Register_7                           := TO_DINT(_dword);

            _dword.%B3                                              := _data[32];
            _dword.%B2                                              := _data[33];
            _dword.%B1                                              := _data[34];
            _dword.%B0                                              := _data[35];
            Inputs.Inputs.Ints.Register_8                           := TO_DINT(_dword);

            _dword.%B3                                              := _data[36];
            _dword.%B2                                              := _data[37];
            _dword.%B1                                              := _data[38];
            _dword.%B0                                              := _data[39];
            Inputs.Inputs.Ints.Register_9                           := TO_DINT(_dword);

            _dword.%B3                                              := _data[40];
            _dword.%B2                                              := _data[41];
            _dword.%B1                                              := _data[42];
            _dword.%B0                                              := _data[43];
            Inputs.Inputs.Ints.Register_10                          := TO_DINT(_dword);

            _dword.%B3                                              := _data[44];
            _dword.%B2                                              := _data[45];
            _dword.%B1                                              := _data[46];
            _dword.%B0                                              := _data[47];
            Inputs.Inputs.Ints.Register_11                          := TO_DINT(_dword);

            _dword.%B3                                              := _data[48];
            _dword.%B2                                              := _data[49];
            _dword.%B1                                              := _data[50];
            _dword.%B0                                              := _data[51];
            Inputs.Inputs.Ints.Register_12                          := TO_DINT(_dword);

            _dword.%B3                                              := _data[52];
            _dword.%B2                                              := _data[53];
            _dword.%B1                                              := _data[54];
            _dword.%B0                                              := _data[55];
            Inputs.Inputs.Ints.Register_13                          := TO_DINT(_dword);

            _dword.%B3                                              := _data[56];
            _dword.%B2                                              := _data[57];
            _dword.%B1                                              := _data[58];
            _dword.%B0                                              := _data[59];
            Inputs.Inputs.Ints.Register_14                          := TO_DINT(_dword);

            _dword.%B3                                              := _data[60];
            _dword.%B2                                              := _data[61];
            _dword.%B1                                              := _data[62];
            _dword.%B0                                              := _data[63];
            Inputs.Inputs.Ints.Register_15                          := TO_DINT(_dword);

            _dword.%B3                                              := _data[64];
            _dword.%B2                                              := _data[65];
            _dword.%B1                                              := _data[66];
            _dword.%B0                                              := _data[67];
            Inputs.Inputs.Ints.Register_16                          := TO_DINT(_dword);

            _dword.%B3                                              := _data[68];
            _dword.%B2                                              := _data[69];
            _dword.%B1                                              := _data[70];
            _dword.%B0                                              := _data[71];
            Inputs.Inputs.Ints.Register_17                          := TO_DINT(_dword);

            _dword.%B3                                              := _data[72];
            _dword.%B2                                              := _data[73];
            _dword.%B1                                              := _data[74];
            _dword.%B0                                              := _data[75];
            Inputs.Inputs.Ints.Register_18                          := TO_DINT(_dword);

            _dword.%B3                                              := _data[76];
            _dword.%B2                                              := _data[77];
            _dword.%B1                                              := _data[78];
            _dword.%B0                                              := _data[79];
            Inputs.Inputs.Ints.Register_19                          := TO_DINT(_dword);

            _dword.%B3                                              := _data[80];
            _dword.%B2                                              := _data[81];
            _dword.%B1                                              := _data[82];
            _dword.%B0                                              := _data[83];
            Inputs.Inputs.Ints.Register_20                          := TO_DINT(_dword);

            _dword.%B3                                              := _data[84];
            _dword.%B2                                              := _data[85];
            _dword.%B1                                              := _data[86];
            _dword.%B0                                              := _data[87];
            Inputs.Inputs.Ints.Register_21                          := TO_DINT(_dword);

            _dword.%B3                                              := _data[88];
            _dword.%B2                                              := _data[89];
            _dword.%B1                                              := _data[90];
            _dword.%B0                                              := _data[91];
            Inputs.Inputs.Ints.Register_22                          := TO_DINT(_dword);

            _dword.%B3                                              := _data[92];
            _dword.%B2                                              := _data[93];
            _dword.%B1                                              := _data[94];
            _dword.%B0                                              := _data[95];
            Inputs.Inputs.Ints.Register_23                          := TO_DINT(_dword);

            //INPUTS T20 BITS => st_URO_CB3_T2OFloatRegsData
            _retVal := Siemens.Simatic.DistributedIO.ReadData((Config.HWIDs.HwId_AxoUrRobotics_T2O_General_Purpose_Float_Registers), _data);
            IF _retVal > WORD#0 THEN
                Messenger.Activate(UINT#1207, eAxoMessageCategory#Error);
                Status.Error.Id := UINT#1207;
                RETURN;
            END_IF;
            _dword.%B3                                              := _data[0];
            _dword.%B2                                              := _data[1];
            _dword.%B1                                              := _data[2];
            _dword.%B0                                              := _data[3];
            Inputs.Inputs.Floats.Register_0                         := TO_REAL(_dword);

            _dword.%B3                                              := _data[4];
            _dword.%B2                                              := _data[5];
            _dword.%B1                                              := _data[6];
            _dword.%B0                                              := _data[7];
            Inputs.Inputs.Floats.Register_1                         := TO_REAL(_dword);

            _dword.%B3                                              := _data[8];
            _dword.%B2                                              := _data[9];
            _dword.%B1                                              := _data[10];
            _dword.%B0                                              := _data[11];
            Inputs.Inputs.Floats.Register_2                         := TO_REAL(_dword);

            _dword.%B3                                              := _data[12];
            _dword.%B2                                              := _data[13];
            _dword.%B1                                              := _data[14];
            _dword.%B0                                              := _data[15];
            Inputs.Inputs.Floats.Register_3                         := TO_REAL(_dword);

            _dword.%B3                                              := _data[16];
            _dword.%B2                                              := _data[17];
            _dword.%B1                                              := _data[18];
            _dword.%B0                                              := _data[19];
            Inputs.Inputs.Floats.Register_4                         := TO_REAL(_dword);

            _dword.%B3                                              := _data[20];
            _dword.%B2                                              := _data[21];
            _dword.%B1                                              := _data[22];
            _dword.%B0                                              := _data[23];
            Inputs.Inputs.Floats.Register_5                         := TO_REAL(_dword);

            _dword.%B3                                              := _data[24];
            _dword.%B2                                              := _data[25];
            _dword.%B1                                              := _data[26];
            _dword.%B0                                              := _data[27];
            Inputs.Inputs.Floats.Register_6                         := TO_REAL(_dword);

            _dword.%B3                                              := _data[28];
            _dword.%B2                                              := _data[29];
            _dword.%B1                                              := _data[30];
            _dword.%B0                                              := _data[31];
            Inputs.Inputs.Floats.Register_7                         := TO_REAL(_dword);

            _dword.%B3                                              := _data[32];
            _dword.%B2                                              := _data[33];
            _dword.%B1                                              := _data[34];
            _dword.%B0                                              := _data[35];
            Inputs.Inputs.Floats.Register_8                         := TO_REAL(_dword);

            _dword.%B3                                              := _data[36];
            _dword.%B2                                              := _data[37];
            _dword.%B1                                              := _data[38];
            _dword.%B0                                              := _data[39];
            Inputs.Inputs.Floats.Register_9                         := TO_REAL(_dword);

            _dword.%B3                                              := _data[40];
            _dword.%B2                                              := _data[41];
            _dword.%B1                                              := _data[42];
            _dword.%B0                                              := _data[43];
            Inputs.Inputs.Floats.Register_10                        := TO_REAL(_dword);

            _dword.%B3                                              := _data[44];
            _dword.%B2                                              := _data[45];
            _dword.%B1                                              := _data[46];
            _dword.%B0                                              := _data[47];
            Inputs.Inputs.Floats.Register_11                        := TO_REAL(_dword);

            _dword.%B3                                              := _data[48];
            _dword.%B2                                              := _data[49];
            _dword.%B1                                              := _data[50];
            _dword.%B0                                              := _data[51];
            Inputs.Inputs.Floats.Register_12                        := TO_REAL(_dword);

            _dword.%B3                                              := _data[52];
            _dword.%B2                                              := _data[53];
            _dword.%B1                                              := _data[54];
            _dword.%B0                                              := _data[55];
            Inputs.Inputs.Floats.Register_13                        := TO_REAL(_dword);

            _dword.%B3                                              := _data[56];
            _dword.%B2                                              := _data[57];
            _dword.%B1                                              := _data[58];
            _dword.%B0                                              := _data[59];
            Inputs.Inputs.Floats.Register_14                        := TO_REAL(_dword);

            _dword.%B3                                              := _data[60];
            _dword.%B2                                              := _data[61];
            _dword.%B1                                              := _data[62];
            _dword.%B0                                              := _data[63];
            Inputs.Inputs.Floats.Register_15                        := TO_REAL(_dword);

            _dword.%B3                                              := _data[64];
            _dword.%B2                                              := _data[65];
            _dword.%B1                                              := _data[66];
            _dword.%B0                                              := _data[67];
            Inputs.Inputs.Floats.Register_16                        := TO_REAL(_dword);

            _dword.%B3                                              := _data[68];
            _dword.%B2                                              := _data[69];
            _dword.%B1                                              := _data[70];
            _dword.%B0                                              := _data[71];
            Inputs.Inputs.Floats.Register_17                        := TO_REAL(_dword);

            _dword.%B3                                              := _data[72];
            _dword.%B2                                              := _data[73];
            _dword.%B1                                              := _data[74];
            _dword.%B0                                              := _data[75];
            Inputs.Inputs.Floats.Register_18                        := TO_REAL(_dword);

            _dword.%B3                                              := _data[76];
            _dword.%B2                                              := _data[77];
            _dword.%B1                                              := _data[78];
            _dword.%B0                                              := _data[79];
            Inputs.Inputs.Floats.Register_19                        := TO_REAL(_dword);

            _dword.%B3                                              := _data[80];
            _dword.%B2                                              := _data[81];
            _dword.%B1                                              := _data[82];
            _dword.%B0                                              := _data[83];
            Inputs.Inputs.Floats.Register_20                        := TO_REAL(_dword);

            _dword.%B3                                              := _data[84];
            _dword.%B2                                              := _data[85];
            _dword.%B1                                              := _data[86];
            _dword.%B0                                              := _data[87];
            Inputs.Inputs.Floats.Register_21                        := TO_REAL(_dword);

            _dword.%B3                                              := _data[88];
            _dword.%B2                                              := _data[89];
            _dword.%B1                                              := _data[90];
            _dword.%B0                                              := _data[91];
            Inputs.Inputs.Floats.Register_22                        := TO_REAL(_dword);

            _dword.%B3                                              := _data[92];
            _dword.%B2                                              := _data[93];
            _dword.%B1                                              := _data[94];
            _dword.%B0                                              := _data[95];
            Inputs.Inputs.Floats.Register_23                        := TO_REAL(_dword);

             Inputs.RobotMode := THIS.GetRobotModeDescription(Inputs.Inputs.Robot.RobotMode);
            //SYSTEM INPUTS
            //Area/positions flags this  should be obsolete because Zones and InPosition is used as byte below
            Inputs.InArea_1                                         := Inputs.Inputs.Bits.Register_0;
            Inputs.InArea_2                                         := Inputs.Inputs.Bits.Register_1;
            Inputs.InArea_3                                         := Inputs.Inputs.Bits.Register_2;
            Inputs.InArea_4                                         := Inputs.Inputs.Bits.Register_3;
            Inputs.InPosition_1                                     := Inputs.Inputs.Bits.Register_4;
            Inputs.InPosition_2                                     := Inputs.Inputs.Bits.Register_5;
            Inputs.InPosition_3                                     := Inputs.Inputs.Bits.Register_6;
            Inputs.InPosition_4                                     := Inputs.Inputs.Bits.Register_7;

            //Tool signals

            Inputs.Tool_1_Retract                                   := Inputs.Inputs.Bits.Register_8;
            Inputs.Tool_1_Extend                                    := Inputs.Inputs.Bits.Register_9;
            Inputs.Tool_2_Retract                                   := Inputs.Inputs.Bits.Register_10;
            Inputs.Tool_2_Extend                                    := Inputs.Inputs.Bits.Register_11;
            Inputs.Tool_3_Retract                                   := Inputs.Inputs.Bits.Register_12;
            Inputs.Tool_3_Extend                                    := Inputs.Inputs.Bits.Register_13;
            Inputs.Tool_4_Retract                                   := Inputs.Inputs.Bits.Register_14;
            Inputs.Tool_4_Extend                                    := Inputs.Inputs.Bits.Register_15;
